// TIA Portal V17 export
VAR_GLOBAL   // PLC tag table "MyTagTableWithConsts"
   MyTag AT %I1.1 : Bool;
   "MyWeird%Tag" AT %I1.2 : Bool;
END_VAR
VAR_GLOBAL CONSTANT   // user constants
   MyConst : Bool := True;
   "MyWeird%Const" : Bool := False;
   MyConstWithComment : Bool := True;   // This is my comment
END_VAR
